INTERFACE I_Drive

{attribute 'monitoring':='call'}
PROPERTY Active : BOOL
GET
END_GET
END_PROPERTY

{attribute 'monitoring':='call'}
PROPERTY AtHome : BOOL
GET
END_GET
END_PROPERTY

{attribute 'monitoring':='call'}
PROPERTY Error : BOOL
GET
END_GET
END_PROPERTY

{attribute 'monitoring':='call'}
PROPERTY HomeSet : BOOL
GET
END_GET
END_PROPERTY

METHOD ABSTRACT homingSequence : BOOL
VAR_INPUT
END_VAR
END_METHOD

METHOD reset : BOOL
VAR_INPUT
END_VAR
END_METHOD

METHOD ABSTRACT stop : BOOL
VAR_INPUT
END_VAR
END_METHOD

METHOD toHome : BOOL
VAR_INPUT
END_VAR
END_METHOD

END_INTERFACE

(* stored: Version 1.1.0.1, ProductVersion 3.1.4024.11
   Itf I_Drive: Id {e1eb8c48-7b7b-492d-8b70-2ec679581052}
   Property Active: Id {b9f317c0-8d70-497e-b1c4-c9ce1c341d8c}
   Get Get: Id {542f606a-6965-47b8-a90c-0987a4a5aa56}
   Property AtHome: Id {d3367613-6051-45a7-bb4e-d3da08972b02}
   Get Get: Id {f5833afb-75b8-4951-b479-709ca6d37d41}
   Property Error: Id {bfa5fc42-6272-44a8-97a1-4e16bed4ae67}
   Get Get: Id {75b7eae4-04ec-4db9-9a80-1f0807ffbf1f}
   Property HomeSet: Id {55d8d979-3411-4a92-89a3-450c116ac487}
   Get Get: Id {aba12fc3-cb14-4795-b287-e75716726c36}
   Method homingSequence: Id {e3fa5096-da88-4f84-a6d1-7c42475dba98}
   Method reset: Id {da53779b-f00e-4ac0-b5e4-28f6bb658428}
   Method stop: Id {29a7ef21-dfdd-4749-92df-d8e96ac6dd6b}
   Method toHome: Id {d43fb5d5-cefa-4cbf-b294-d8f59083e287} *)
